// TIA Portal V20 export
ORGANIZATION_BLOCK "Startup"   // OB100, LAD, Startup
TITLE = "Complete Restart"
// stored: AutoNumber false, IsIECCheckEnabled true, SetENOAutomatically true
   VAR_INPUT
      LostRetentive : Bool;   // True if retentive data are lost
      LostRTC : Bool;   // True if date and time are lost
   END_VAR
   VAR_TEMP
      tempError : Bool;
      tempStatus : Word;
      tempDiagnostics : "LAF_typeDiagnosticsSimple";
   END_VAR
BEGIN

REGION Network 1: Erster Zyklus bit setzen / Set first cycle bit
   // Setze das "erster Zyklus" Signal und die Signale immer EIN sowie immer AUS / Set the first cycle signal
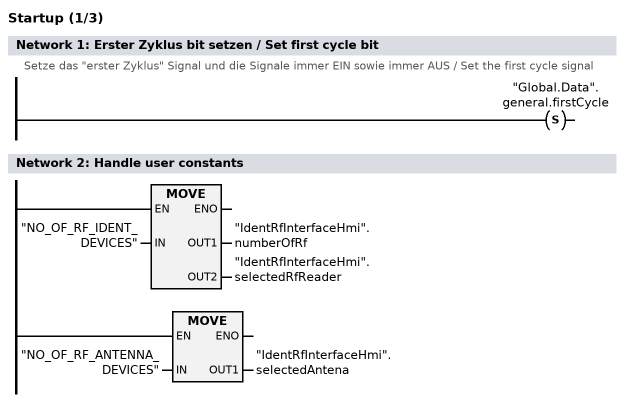
   RUNG wire#powerrail
      S_Coil( "Global.Data".general.firstCycle )
   END_RUNG
   // the same network as SCL:
   "Global.Data".general.firstCycle := TRUE;
END_REGION

REGION Network 2: Handle user constants
   RUNG wire#powerrail
      Move(in := "NO_OF_RF_IDENT_DEVICES", out1 => "IdentRfInterfaceHmi".numberOfRf, out2 => "IdentRfInterfaceHmi".selectedRfReader)
   END_RUNG
   RUNG wire#powerrail
      Move(in := "NO_OF_RF_ANTENNA_DEVICES", out1 => "IdentRfInterfaceHmi".selectedAntena)
   END_RUNG
   // the same network as SCL:
   "IdentRfInterfaceHmi".numberOfRf := "NO_OF_RF_IDENT_DEVICES";
   "IdentRfInterfaceHmi".selectedRfReader := "NO_OF_RF_IDENT_DEVICES";
   "IdentRfInterfaceHmi".selectedAntena := "NO_OF_RF_ANTENNA_DEVICES";
END_REGION

REGION Network 3: Set drive objects for drive diagnostic
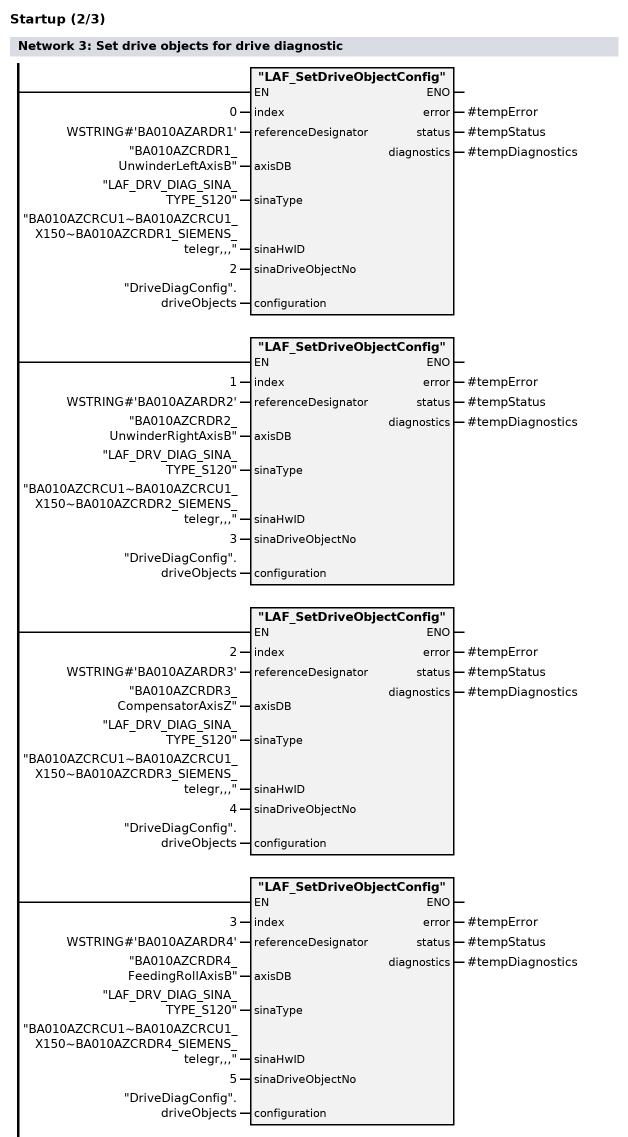
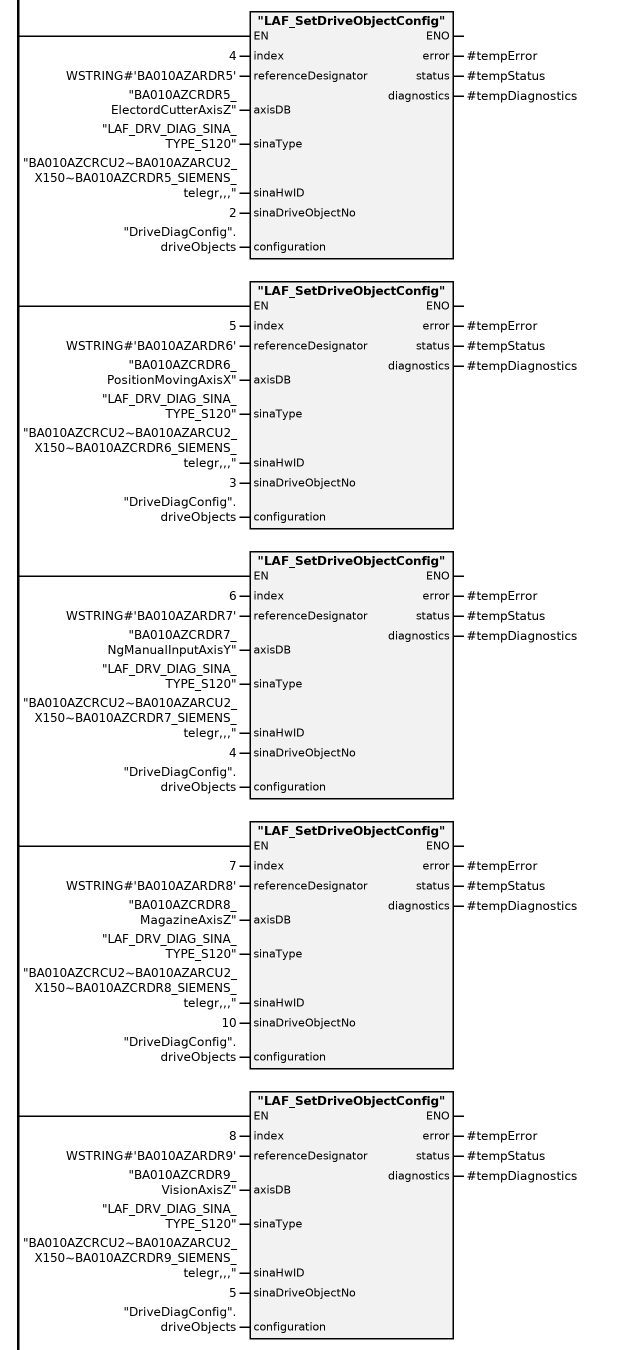
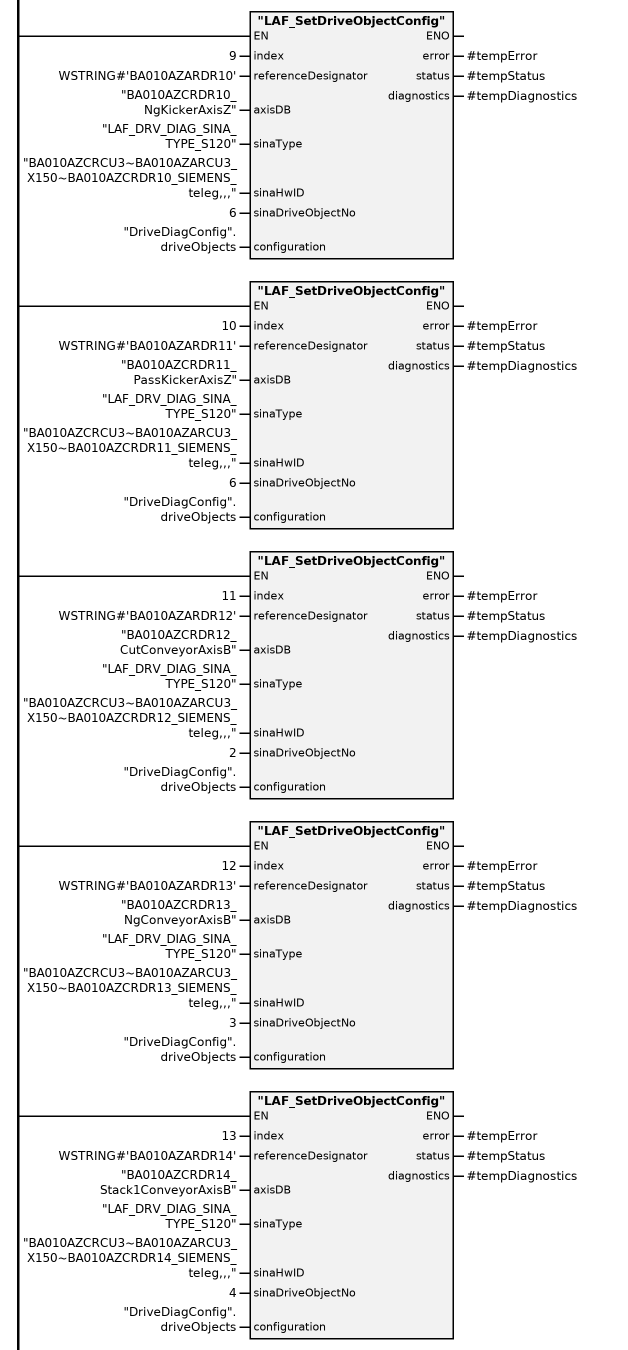
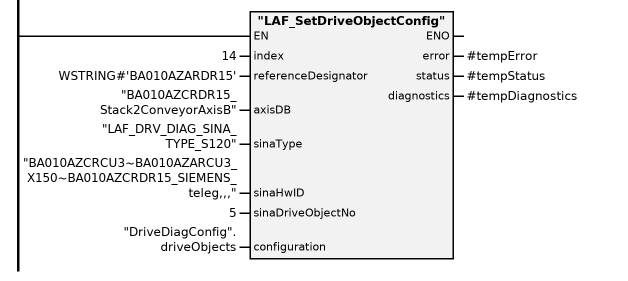
   RUNG wire#powerrail
      "LAF_SetDriveObjectConfig"(index := 0, referenceDesignator := WSTRING#'BA010AZARDR1', axisDB := "BA010AZCRDR1_UnwinderLeftAxisB", sinaType := "LAF_DRV_DIAG_SINA_TYPE_S120", sinaHwID := "BA010AZCRCU1~BA010AZCRCU1_X150~BA010AZCRDR1_SIEMENS_telegr,,,", sinaDriveObjectNo := 2, configuration := "DriveDiagConfig".driveObjects, error => #tempError, status => #tempStatus, diagnostics => #tempDiagnostics)
   END_RUNG
   RUNG wire#powerrail
      "LAF_SetDriveObjectConfig"(index := 1, referenceDesignator := WSTRING#'BA010AZARDR2', axisDB := "BA010AZCRDR2_UnwinderRightAxisB", sinaType := "LAF_DRV_DIAG_SINA_TYPE_S120", sinaHwID := "BA010AZCRCU1~BA010AZCRCU1_X150~BA010AZCRDR2_SIEMENS_telegr,,,", sinaDriveObjectNo := 3, configuration := "DriveDiagConfig".driveObjects, error => #tempError, status => #tempStatus, diagnostics => #tempDiagnostics)
   END_RUNG
   RUNG wire#powerrail
      "LAF_SetDriveObjectConfig"(index := 2, referenceDesignator := WSTRING#'BA010AZARDR3', axisDB := "BA010AZCRDR3_CompensatorAxisZ", sinaType := "LAF_DRV_DIAG_SINA_TYPE_S120", sinaHwID := "BA010AZCRCU1~BA010AZCRCU1_X150~BA010AZCRDR3_SIEMENS_telegr,,,", sinaDriveObjectNo := 4, configuration := "DriveDiagConfig".driveObjects, error => #tempError, status => #tempStatus, diagnostics => #tempDiagnostics)
   END_RUNG
   RUNG wire#powerrail
      "LAF_SetDriveObjectConfig"(index := 3, referenceDesignator := WSTRING#'BA010AZARDR4', axisDB := "BA010AZCRDR4_FeedingRollAxisB", sinaType := "LAF_DRV_DIAG_SINA_TYPE_S120", sinaHwID := "BA010AZCRCU1~BA010AZCRCU1_X150~BA010AZCRDR4_SIEMENS_telegr,,,", sinaDriveObjectNo := 5, configuration := "DriveDiagConfig".driveObjects, error => #tempError, status => #tempStatus, diagnostics => #tempDiagnostics)
   END_RUNG
   RUNG wire#powerrail
      "LAF_SetDriveObjectConfig"(index := 4, referenceDesignator := WSTRING#'BA010AZARDR5', axisDB := "BA010AZCRDR5_ElectordCutterAxisZ", sinaType := "LAF_DRV_DIAG_SINA_TYPE_S120", sinaHwID := "BA010AZCRCU2~BA010AZARCU2_X150~BA010AZCRDR5_SIEMENS_telegr,,,", sinaDriveObjectNo := 2, configuration := "DriveDiagConfig".driveObjects, error => #tempError, status => #tempStatus, diagnostics => #tempDiagnostics)
   END_RUNG
   RUNG wire#powerrail
      "LAF_SetDriveObjectConfig"(index := 5, referenceDesignator := WSTRING#'BA010AZARDR6', axisDB := "BA010AZCRDR6_PositionMovingAxisX", sinaType := "LAF_DRV_DIAG_SINA_TYPE_S120", sinaHwID := "BA010AZCRCU2~BA010AZARCU2_X150~BA010AZCRDR6_SIEMENS_telegr,,,", sinaDriveObjectNo := 3, configuration := "DriveDiagConfig".driveObjects, error => #tempError, status => #tempStatus, diagnostics => #tempDiagnostics)
   END_RUNG
   RUNG wire#powerrail
      "LAF_SetDriveObjectConfig"(index := 6, referenceDesignator := WSTRING#'BA010AZARDR7', axisDB := "BA010AZCRDR7_NgManualInputAxisY", sinaType := "LAF_DRV_DIAG_SINA_TYPE_S120", sinaHwID := "BA010AZCRCU2~BA010AZARCU2_X150~BA010AZCRDR7_SIEMENS_telegr,,,", sinaDriveObjectNo := 4, configuration := "DriveDiagConfig".driveObjects, error => #tempError, status => #tempStatus, diagnostics => #tempDiagnostics)
   END_RUNG
   RUNG wire#powerrail
      "LAF_SetDriveObjectConfig"(index := 7, referenceDesignator := WSTRING#'BA010AZARDR8', axisDB := "BA010AZCRDR8_MagazineAxisZ", sinaType := "LAF_DRV_DIAG_SINA_TYPE_S120", sinaHwID := "BA010AZCRCU2~BA010AZARCU2_X150~BA010AZCRDR8_SIEMENS_telegr,,,", sinaDriveObjectNo := 10, configuration := "DriveDiagConfig".driveObjects, error => #tempError, status => #tempStatus, diagnostics => #tempDiagnostics)
   END_RUNG
   RUNG wire#powerrail
      "LAF_SetDriveObjectConfig"(index := 8, referenceDesignator := WSTRING#'BA010AZARDR9', axisDB := "BA010AZCRDR9_VisionAxisZ", sinaType := "LAF_DRV_DIAG_SINA_TYPE_S120", sinaHwID := "BA010AZCRCU2~BA010AZARCU2_X150~BA010AZCRDR9_SIEMENS_telegr,,,", sinaDriveObjectNo := 5, configuration := "DriveDiagConfig".driveObjects, error => #tempError, status => #tempStatus, diagnostics => #tempDiagnostics)
   END_RUNG
   RUNG wire#powerrail
      "LAF_SetDriveObjectConfig"(index := 9, referenceDesignator := WSTRING#'BA010AZARDR10', axisDB := "BA010AZCRDR10_NgKickerAxisZ", sinaType := "LAF_DRV_DIAG_SINA_TYPE_S120", sinaHwID := "BA010AZCRCU3~BA010AZARCU3_X150~BA010AZCRDR10_SIEMENS_teleg,,,", sinaDriveObjectNo := 6, configuration := "DriveDiagConfig".driveObjects, error => #tempError, status => #tempStatus, diagnostics => #tempDiagnostics)
   END_RUNG
   RUNG wire#powerrail
      "LAF_SetDriveObjectConfig"(index := 10, referenceDesignator := WSTRING#'BA010AZARDR11', axisDB := "BA010AZCRDR11_PassKickerAxisZ", sinaType := "LAF_DRV_DIAG_SINA_TYPE_S120", sinaHwID := "BA010AZCRCU3~BA010AZARCU3_X150~BA010AZCRDR11_SIEMENS_teleg,,,", sinaDriveObjectNo := 6, configuration := "DriveDiagConfig".driveObjects, error => #tempError, status => #tempStatus, diagnostics => #tempDiagnostics)
   END_RUNG
   RUNG wire#powerrail
      "LAF_SetDriveObjectConfig"(index := 11, referenceDesignator := WSTRING#'BA010AZARDR12', axisDB := "BA010AZCRDR12_CutConveyorAxisB", sinaType := "LAF_DRV_DIAG_SINA_TYPE_S120", sinaHwID := "BA010AZCRCU3~BA010AZARCU3_X150~BA010AZCRDR12_SIEMENS_teleg,,,", sinaDriveObjectNo := 2, configuration := "DriveDiagConfig".driveObjects, error => #tempError, status => #tempStatus, diagnostics => #tempDiagnostics)
   END_RUNG
   RUNG wire#powerrail
      "LAF_SetDriveObjectConfig"(index := 12, referenceDesignator := WSTRING#'BA010AZARDR13', axisDB := "BA010AZCRDR13_NgConveyorAxisB", sinaType := "LAF_DRV_DIAG_SINA_TYPE_S120", sinaHwID := "BA010AZCRCU3~BA010AZARCU3_X150~BA010AZCRDR13_SIEMENS_teleg,,,", sinaDriveObjectNo := 3, configuration := "DriveDiagConfig".driveObjects, error => #tempError, status => #tempStatus, diagnostics => #tempDiagnostics)
   END_RUNG
   RUNG wire#powerrail
      "LAF_SetDriveObjectConfig"(index := 13, referenceDesignator := WSTRING#'BA010AZARDR14', axisDB := "BA010AZCRDR14_Stack1ConveyorAxisB", sinaType := "LAF_DRV_DIAG_SINA_TYPE_S120", sinaHwID := "BA010AZCRCU3~BA010AZARCU3_X150~BA010AZCRDR14_SIEMENS_teleg,,,", sinaDriveObjectNo := 4, configuration := "DriveDiagConfig".driveObjects, error => #tempError, status => #tempStatus, diagnostics => #tempDiagnostics)
   END_RUNG
   RUNG wire#powerrail
      "LAF_SetDriveObjectConfig"(index := 14, referenceDesignator := WSTRING#'BA010AZARDR15', axisDB := "BA010AZCRDR15_Stack2ConveyorAxisB", sinaType := "LAF_DRV_DIAG_SINA_TYPE_S120", sinaHwID := "BA010AZCRCU3~BA010AZARCU3_X150~BA010AZCRDR15_SIEMENS_teleg,,,", sinaDriveObjectNo := 5, configuration := "DriveDiagConfig".driveObjects, error => #tempError, status => #tempStatus, diagnostics => #tempDiagnostics)
   END_RUNG
   // the same network as SCL:
   "LAF_SetDriveObjectConfig"(index := 0,
                           referenceDesignator := WSTRING#'BA010AZARDR1',
                           axisDB := "BA010AZCRDR1_UnwinderLeftAxisB",
                           sinaType := "LAF_DRV_DIAG_SINA_TYPE_S120",
                           sinaHwID := "BA010AZCRCU1~BA010AZCRCU1_X150~BA010AZCRDR1_SIEMENS_telegr,,,",
                           sinaDriveObjectNo := 2,
                           configuration := "DriveDiagConfig".driveObjects,
                           error => #tempError,
                           status => #tempStatus,
                           diagnostics => #tempDiagnostics);
   "LAF_SetDriveObjectConfig"(index := 1,
                           referenceDesignator := WSTRING#'BA010AZARDR2',
                           axisDB := "BA010AZCRDR2_UnwinderRightAxisB",
                           sinaType := "LAF_DRV_DIAG_SINA_TYPE_S120",
                           sinaHwID := "BA010AZCRCU1~BA010AZCRCU1_X150~BA010AZCRDR2_SIEMENS_telegr,,,",
                           sinaDriveObjectNo := 3,
                           configuration := "DriveDiagConfig".driveObjects,
                           error => #tempError,
                           status => #tempStatus,
                           diagnostics => #tempDiagnostics);
   "LAF_SetDriveObjectConfig"(index := 2,
                           referenceDesignator := WSTRING#'BA010AZARDR3',
                           axisDB := "BA010AZCRDR3_CompensatorAxisZ",
                           sinaType := "LAF_DRV_DIAG_SINA_TYPE_S120",
                           sinaHwID := "BA010AZCRCU1~BA010AZCRCU1_X150~BA010AZCRDR3_SIEMENS_telegr,,,",
                           sinaDriveObjectNo := 4,
                           configuration := "DriveDiagConfig".driveObjects,
                           error => #tempError,
                           status => #tempStatus,
                           diagnostics => #tempDiagnostics);
   "LAF_SetDriveObjectConfig"(index := 3,
                           referenceDesignator := WSTRING#'BA010AZARDR4',
                           axisDB := "BA010AZCRDR4_FeedingRollAxisB",
                           sinaType := "LAF_DRV_DIAG_SINA_TYPE_S120",
                           sinaHwID := "BA010AZCRCU1~BA010AZCRCU1_X150~BA010AZCRDR4_SIEMENS_telegr,,,",
                           sinaDriveObjectNo := 5,
                           configuration := "DriveDiagConfig".driveObjects,
                           error => #tempError,
                           status => #tempStatus,
                           diagnostics => #tempDiagnostics);
   "LAF_SetDriveObjectConfig"(index := 4,
                           referenceDesignator := WSTRING#'BA010AZARDR5',
                           axisDB := "BA010AZCRDR5_ElectordCutterAxisZ",
                           sinaType := "LAF_DRV_DIAG_SINA_TYPE_S120",
                           sinaHwID := "BA010AZCRCU2~BA010AZARCU2_X150~BA010AZCRDR5_SIEMENS_telegr,,,",
                           sinaDriveObjectNo := 2,
                           configuration := "DriveDiagConfig".driveObjects,
                           error => #tempError,
                           status => #tempStatus,
                           diagnostics => #tempDiagnostics);
   "LAF_SetDriveObjectConfig"(index := 5,
                           referenceDesignator := WSTRING#'BA010AZARDR6',
                           axisDB := "BA010AZCRDR6_PositionMovingAxisX",
                           sinaType := "LAF_DRV_DIAG_SINA_TYPE_S120",
                           sinaHwID := "BA010AZCRCU2~BA010AZARCU2_X150~BA010AZCRDR6_SIEMENS_telegr,,,",
                           sinaDriveObjectNo := 3,
                           configuration := "DriveDiagConfig".driveObjects,
                           error => #tempError,
                           status => #tempStatus,
                           diagnostics => #tempDiagnostics);
   "LAF_SetDriveObjectConfig"(index := 6,
                           referenceDesignator := WSTRING#'BA010AZARDR7',
                           axisDB := "BA010AZCRDR7_NgManualInputAxisY",
                           sinaType := "LAF_DRV_DIAG_SINA_TYPE_S120",
                           sinaHwID := "BA010AZCRCU2~BA010AZARCU2_X150~BA010AZCRDR7_SIEMENS_telegr,,,",
                           sinaDriveObjectNo := 4,
                           configuration := "DriveDiagConfig".driveObjects,
                           error => #tempError,
                           status => #tempStatus,
                           diagnostics => #tempDiagnostics);
   "LAF_SetDriveObjectConfig"(index := 7,
                           referenceDesignator := WSTRING#'BA010AZARDR8',
                           axisDB := "BA010AZCRDR8_MagazineAxisZ",
                           sinaType := "LAF_DRV_DIAG_SINA_TYPE_S120",
                           sinaHwID := "BA010AZCRCU2~BA010AZARCU2_X150~BA010AZCRDR8_SIEMENS_telegr,,,",
                           sinaDriveObjectNo := 10,
                           configuration := "DriveDiagConfig".driveObjects,
                           error => #tempError,
                           status => #tempStatus,
                           diagnostics => #tempDiagnostics);
   "LAF_SetDriveObjectConfig"(index := 8,
                           referenceDesignator := WSTRING#'BA010AZARDR9',
                           axisDB := "BA010AZCRDR9_VisionAxisZ",
                           sinaType := "LAF_DRV_DIAG_SINA_TYPE_S120",
                           sinaHwID := "BA010AZCRCU2~BA010AZARCU2_X150~BA010AZCRDR9_SIEMENS_telegr,,,",
                           sinaDriveObjectNo := 5,
                           configuration := "DriveDiagConfig".driveObjects,
                           error => #tempError,
                           status => #tempStatus,
                           diagnostics => #tempDiagnostics);
   "LAF_SetDriveObjectConfig"(index := 9,
                           referenceDesignator := WSTRING#'BA010AZARDR10',
                           axisDB := "BA010AZCRDR10_NgKickerAxisZ",
                           sinaType := "LAF_DRV_DIAG_SINA_TYPE_S120",
                           sinaHwID := "BA010AZCRCU3~BA010AZARCU3_X150~BA010AZCRDR10_SIEMENS_teleg,,,",
                           sinaDriveObjectNo := 6,
                           configuration := "DriveDiagConfig".driveObjects,
                           error => #tempError,
                           status => #tempStatus,
                           diagnostics => #tempDiagnostics);
   "LAF_SetDriveObjectConfig"(index := 10,
                           referenceDesignator := WSTRING#'BA010AZARDR11',
                           axisDB := "BA010AZCRDR11_PassKickerAxisZ",
                           sinaType := "LAF_DRV_DIAG_SINA_TYPE_S120",
                           sinaHwID := "BA010AZCRCU3~BA010AZARCU3_X150~BA010AZCRDR11_SIEMENS_teleg,,,",
                           sinaDriveObjectNo := 6,
                           configuration := "DriveDiagConfig".driveObjects,
                           error => #tempError,
                           status => #tempStatus,
                           diagnostics => #tempDiagnostics);
   "LAF_SetDriveObjectConfig"(index := 11,
                           referenceDesignator := WSTRING#'BA010AZARDR12',
                           axisDB := "BA010AZCRDR12_CutConveyorAxisB",
                           sinaType := "LAF_DRV_DIAG_SINA_TYPE_S120",
                           sinaHwID := "BA010AZCRCU3~BA010AZARCU3_X150~BA010AZCRDR12_SIEMENS_teleg,,,",
                           sinaDriveObjectNo := 2,
                           configuration := "DriveDiagConfig".driveObjects,
                           error => #tempError,
                           status => #tempStatus,
                           diagnostics => #tempDiagnostics);
   "LAF_SetDriveObjectConfig"(index := 12,
                           referenceDesignator := WSTRING#'BA010AZARDR13',
                           axisDB := "BA010AZCRDR13_NgConveyorAxisB",
                           sinaType := "LAF_DRV_DIAG_SINA_TYPE_S120",
                           sinaHwID := "BA010AZCRCU3~BA010AZARCU3_X150~BA010AZCRDR13_SIEMENS_teleg,,,",
                           sinaDriveObjectNo := 3,
                           configuration := "DriveDiagConfig".driveObjects,
                           error => #tempError,
                           status => #tempStatus,
                           diagnostics => #tempDiagnostics);
   "LAF_SetDriveObjectConfig"(index := 13,
                           referenceDesignator := WSTRING#'BA010AZARDR14',
                           axisDB := "BA010AZCRDR14_Stack1ConveyorAxisB",
                           sinaType := "LAF_DRV_DIAG_SINA_TYPE_S120",
                           sinaHwID := "BA010AZCRCU3~BA010AZARCU3_X150~BA010AZCRDR14_SIEMENS_teleg,,,",
                           sinaDriveObjectNo := 4,
                           configuration := "DriveDiagConfig".driveObjects,
                           error => #tempError,
                           status => #tempStatus,
                           diagnostics => #tempDiagnostics);
   "LAF_SetDriveObjectConfig"(index := 14,
                           referenceDesignator := WSTRING#'BA010AZARDR15',
                           axisDB := "BA010AZCRDR15_Stack2ConveyorAxisB",
                           sinaType := "LAF_DRV_DIAG_SINA_TYPE_S120",
                           sinaHwID := "BA010AZCRCU3~BA010AZARCU3_X150~BA010AZCRDR15_SIEMENS_teleg,,,",
                           sinaDriveObjectNo := 5,
                           configuration := "DriveDiagConfig".driveObjects,
                           error => #tempError,
                           status => #tempStatus,
                           diagnostics => #tempDiagnostics);
END_REGION

REGION Network 4: Manual Operation Line
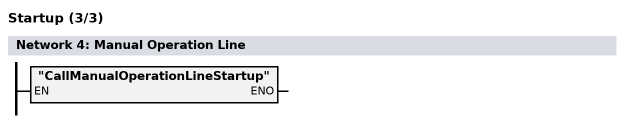
   RUNG wire#powerrail
      "CallManualOperationLineStartup"()
   END_RUNG
   // the same network as SCL:
   "CallManualOperationLineStartup"();
END_REGION
END_ORGANIZATION_BLOCK
